PROGRAM Process_Logging
VAR
END_VAR

//IO0.fb_TimeStamp() ;
device_rtrig() ;

IF IO_Logs.bStart.Q THEN
	IO.LogProcess(	sLogEvent	 := MSG.EVENT_BTN, 
	 				sLogComp	 := MSG.COMP_START, 
	 				sLogAction	 := MSG.ACTION_START, 
	 				sLogStatus	 := MSG.STATUS_ACK,
	 		 		blogFlag	 := TRUE);
//	IF IO.LogProcess.blog_complete OR IO.LogProcess.blog_error THEN
//		IO.bStart := FALSE;
//	END_IF
END_IF		

IF IO_Logs.bReset.Q THEN
//	IO.LogProcess(	sLogEvent	 := MSG.EVENT_BTN, 
	// 				sLogComp	 := MSG.COMP_RESET, 
	 //				sLogAction	 := MSG.ACTION_RESET, 
	 	//			sLogStatus	 := MSG.STATUS_ACK,
	 		// 		blogFlag	 := TRUE);
END_IF	

//IF IO_Logs.bEstop.Q THEN
//	IO.LogProcess(	sLogEvent	 := MSG.EVENT_BTN, 
//	 				sLogComp	 := MSG.COMP_ESTOP, 
//	 				sLogAction	 := MSG.ACTION_ESTOP, 
//	 				sLogStatus	 := MSG.STATUS_ACK,
//	 		 		blogFlag	 := TRUE);
//END_IF

//IF IO_Logs.bOperational_State.Q THEN
//	IO.LogProcess(	sLogEvent	 := MSG.EVENT_BTN, 
//	 				sLogComp	 := MSG.COMP_ESTOP, 
//	 				sLogAction	 := MSG.ACTION_ESTOP, 
//	 				sLogStatus	 := MSG.STATUS_ACK,
//	 		 		blogFlag	 := TRUE);
//END_IF								

//IF IO_Logs.data_send_flag.Q THEN
//	IO.LogProcess(	sLogEvent	 := MSG.EVENT_PROCESS, 
//	 				sLogComp	 := MSG.COMP_SCANNER, 
//	 				sLogAction	 := MSG.ACTION_SCNR_ON, 
//	 				sLogStatus	 := MSG.STATUS_DONE,
//	 		 		blogFlag	 := TRUE);
//END_IF

END_PROGRAM

(* stored: Version 1.1.0.1, ProductVersion 3.1.4024.12
   POU Process_Logging: Id {87b540dd-6262-40f9-9bec-4100db02f950}, SpecialFunc None *)
